(* CODESYS project mbc_Log4TC.library
   Title: Log4TC
   Version: 0.0.1
   Placeholder: Log4TC
   Company: mbc engineering GmbH

Project tree, tasks and I/O mapping:
  libraries: Base Interfaces, * (System); Tc2_Standard, * (Beckhoff Automation GmbH); Tc2_System, * (Beckhoff Automation GmbH); Tc2_Utilities, * (Beckhoff Automation GmbH)
  API/
    Full/
      function block FB_Logger [ST]: FB_init, LoggerContext
    Simple/
      function F_Log3 [ST]
      function F_Log3L [ST]
      function F_LogA3 [ST]
      function F_LogBuilder [ST]
      function F_LogLA3 [ST]
      interface I_LogBuilder: CreateLog, WithContextInt, WithIntArg, WithLogger, WithStringArg
    data type E_LogLevel
    function F_CallLogTask [ST]
    function F_LogContext [ST]
    interface I_ContextBuilder: Reset, WithInt
  GVLs/
    global variables Config
    global variables Const
    global variables GlobalVariables
  ITFs/
    interface I_LogEntryAdder: AddToLogEntry
  POUs/
    Utils/
      function F_DINT_TO_UINT_MAX [ST]
    function F_InternalLog [ST]
    function block FB_ContextBuilder [CFC]: _AddContext, _Copy, _RemoveContext, _Reset, _WriteByte, _WriteInt, AddToLogEntry, Reset, WithInt
    function block FB_Log4TcTask [CFC]: AddLog, Call, FB_init
    function block FB_LogEntry [CFC]: _BufferRemaining, _Copy, _Reset, _WriteArg, _WriteByte, _WriteDInt, _WriteInt, _WriteLInt, _WriteString, _WriteUDInt, _WriteUInt, AddAnyArg, AddBuffer, AddContext, AddTArg, End, GetBuffer, Start
  program Test [ST]
*)

// API/E_LogLevel
{attribute 'qualified_only'}
{attribute 'strict'}
TYPE E_LogLevel :
(
	eTrace 	:= 0,
	eDebug 	:= 1,
	eInfo	:= 2,
	eWarn	:= 3,
	eError	:= 4,
	eFatal	:= 5
) UINT;
END_TYPE

// GVLs/Config
{attribute 'qualified_only'}
VAR_GLOBAL CONSTANT
	eInternalLog		: E_LogLevel := E_LogLevel.eDebug;	(* min. log level for internal logging. *)
	nBufferLen 			: UINT := 8192;		(* Length of per task log buffer in bytes *)
END_VAR

// GVLs/Const
{attribute 'qualified_only'}
VAR_GLOBAL CONSTANT
	nAdsPort			: UINT := 16150; 
	nLogIndexGrp		: UINT := 1;
	nLogIndexOffs		: UINT := 1;
	
	sGlobalLogger		: STRING := '_GLOBAL_';		(* Global logger name for logger without logger input *)
END_VAR

// GVLs/GlobalVariables
{attribute 'qualified_only'}
VAR_GLOBAL
	aTaskLogger			: ARRAY[1..SIZEOF(TwinCAT_SystemInfoVarList._TaskInfo)/SIZEOF(PlcTaskSystemInfo)] OF FB_Log4TcTask;
END_VAR

// API/Full/FB_Logger
{attribute 'reflection'} 
FUNCTION_BLOCK FB_Logger
VAR_INPUT
	bExecute		: BOOL := TRUE;
	eLogLevel		: E_LogLevel;
	sMessage		: Tc2_System.T_MaxString;
	stArg1			: T_Arg := Tc2_Utilities.EMPTY_ARG_VALUE;
	stArg2			: T_Arg := Tc2_Utilities.EMPTY_ARG_VALUE;
	stArg3			: T_Arg := Tc2_Utilities.EMPTY_ARG_VALUE;
	stArg4			: T_Arg := Tc2_Utilities.EMPTY_ARG_VALUE;
	stArg5			: T_Arg := Tc2_Utilities.EMPTY_ARG_VALUE;	
	stArg6			: T_Arg := Tc2_Utilities.EMPTY_ARG_VALUE;	
	stArg7			: T_Arg := Tc2_Utilities.EMPTY_ARG_VALUE;	
	stArg8			: T_Arg := Tc2_Utilities.EMPTY_ARG_VALUE;	
	stArg9			: T_Arg := Tc2_Utilities.EMPTY_ARG_VALUE;	
	stArg10			: T_Arg := Tc2_Utilities.EMPTY_ARG_VALUE;	
	iContextBuilder	: I_ContextBuilder := 0;	
END_VAR
VAR
    {attribute 'instance-path'} 
    {attribute 'noinit'} // 'log4tc.log4Tc_Tester.MAIN.fbLog' bwz. 'log4tc.log4Tc_Tester.GVL.fbLog'
    sInstancePath	: T_MaxString; 	
	sLogger			: T_MaxString;
	fbLoggerContext	: FB_ContextBuilder;
END_VAR
VAR_TEMP
	fbLogEntry		: FB_LogEntry();
	fbSysTime		: Tc2_System.GETSYSTEMTIME;
	nTimestamp		: LINT;
	pBuffer			: PVOID;
	nBufferCount	: UINT;
	iLogEntryAdder	: I_LogEntryAdder;
END_VAR

IF bExecute THEN
	
	fbLogEntry.Start(
		pLogger		:= ADR(sLogger),
		pMessage 	:= ADR(sMessage),
		eLogLevel	:= eLogLevel,
		nTimeStampPlc := nTimestamp,
		nTimeStampClock := 0
	);
	
	fbLogEntry.AddTArg(1, stArg1);
	fbLogEntry.AddTArg(2, stArg2);
	fbLogEntry.AddTArg(3, stArg3);
	fbLogEntry.AddTArg(4, stArg4);
	fbLogEntry.AddTArg(5, stArg5);
	fbLogEntry.AddTArg(6, stArg6);
	fbLogEntry.AddTArg(7, stArg7);
	fbLogEntry.AddTArg(8, stArg8);
	fbLogEntry.AddTArg(9, stArg9);
	fbLogEntry.AddTArg(10, stArg10);
	
	//IF __QUERYINTERFACE(F_GetTaskContext(), iLogEntryAdder) THEN
		//iLogEntryAdder.AddToLogEntry(fbLogEntry);
	//END_IF
	
	fbLoggerContext.AddToLogEntry(fbLogEntry);
	
	IF iContextBuilder <> 0 AND __QUERYINTERFACE(iContextBuilder, iLogEntryAdder) THEN
		iLogEntryAdder.AddToLogEntry(fbLogEntry);
	END_IF
	
	// TODO instance path
	
	IF fbLogEntry.End() THEN
		// Add to buffer
		fbLogEntry.GetBuffer(
			pBuffer			=> pBuffer,
			nBufferCount	=> nBufferCount
		);
		GlobalVariables.aTaskLogger[GETCURTASKINDEXEX()].AddLog(pBuffer, nBufferCount);
	END_IF
END_IF

// reset arguments to default values
bExecute := TRUE;
stArg1 := Tc2_Utilities.EMPTY_ARG_VALUE;
stArg2 := Tc2_Utilities.EMPTY_ARG_VALUE;
stArg3 := Tc2_Utilities.EMPTY_ARG_VALUE;
stArg4 := Tc2_Utilities.EMPTY_ARG_VALUE;
stArg5 := Tc2_Utilities.EMPTY_ARG_VALUE;
stArg6 := Tc2_Utilities.EMPTY_ARG_VALUE;
stArg7 := Tc2_Utilities.EMPTY_ARG_VALUE;
stArg8 := Tc2_Utilities.EMPTY_ARG_VALUE;
stArg9 := Tc2_Utilities.EMPTY_ARG_VALUE;
stArg10 := Tc2_Utilities.EMPTY_ARG_VALUE;
iContextBuilder := 0;

METHOD FB_init : BOOL
VAR_INPUT
	bInitRetains : BOOL; // if TRUE, the retain variables are initialized (warm start / cold start)
	bInCopyCode : BOOL;  // if TRUE, the instance afterwards gets moved into the copy code (online change)
	sLogger		: T_MaxString;
END_VAR
THIS^.sLogger := sLogger;
END_METHOD

PROPERTY PUBLIC LoggerContext : I_ContextBuilder
GET
LoggerContext := fbLoggerContext;
END_GET
END_PROPERTY

END_FUNCTION_BLOCK

// API/I_ContextBuilder
INTERFACE I_ContextBuilder EXTENDS __System.IQueryInterface

METHOD Reset : I_ContextBuilder
VAR_INPUT
END_VAR
END_METHOD

METHOD WithInt : I_ContextBuilder
VAR_INPUT
	sName		: T_MaxString;
	nValue		: INT;
END_VAR
END_METHOD

END_INTERFACE

// POUs/FB_ContextBuilder
FUNCTION_BLOCK FB_ContextBuilder IMPLEMENTS I_ContextBuilder, I_LogEntryAdder
VAR CONSTANT
	nBufferSize			: UINT := 1024;
END_VAR
VAR
	aBuffer				: ARRAY[0..nBufferSize - 1] OF BYTE;	(* buffer for context variables *)
	nBufferCount		: UINT := 0;
	
	aContext			: ARRAY[0..19] OF UINT;
	nContextCount		: UINT(0..20) := 0;
END_VAR

METHOD PRIVATE _AddContext : BOOL
VAR_INPUT
END_VAR
IF nContextCount < 20 THEN
	aContext[nContextCount] := nBufferCount;
	nContextCount := nContextCount + 1;
	_AddContext := TRUE;
ELSE
	_AddContext := FALSE;
END_IF
END_METHOD

METHOD PRIVATE _Copy : BOOL
VAR_INPUT
	pSrc		: PVOID;
	nCount		: UINT;
END_VAR
IF (nBufferSize - nBufferCount) >= nCount THEN
	MEMCPY(ADR(aBuffer) + nBufferCount, pSrc, nCount);
	nBufferCount := nBufferCount + nCount;
	
	_Copy := TRUE;
ELSE
	_Copy := FALSE;
END_IF
END_METHOD

METHOD PRIVATE _RemoveContext : BOOL
VAR_INPUT
	refName		: REFERENCE TO Tc2_System.T_MaxString;
END_VAR
VAR
	nIdx		: UINT;
	nBufferOff	: UINT;
END_VAR
IF nContextCount > 0 THEN
	FOR nIdx := 0 TO nContextCount - 1 DO
		IF MEMCMP(ADR(refName), ADR(aBuffer) + aContext[nIdx], INT_TO_UDINT(LEN(refName) + 1)) = 0 THEN
			(* Found - remove entry and compact buffer *)
			IF (nIdx + 1) < nContextCount THEN
				// Move buffer data
				MEMMOVE(
					ADR(aBuffer) + aContext[nIdx], 
					ADR(aBuffer) + aContext[nIdx + 1], 
					nBufferCount - aContext[nIdx + 1]
				);
				
				nBufferOff := aContext[nIdx + 1] - aContext[nIdx];
				nBufferCount := nBufferCount - nBufferOff;
				
				// Move and change index
				WHILE (nIdx + 1) < nContextCount DO
					aContext[nIdx] := aContext[nIdx + 1] - nBufferOff;
					nIdx := nIdx + 1;
				END_WHILE
			END_IF

			nContextCount := nContextCount - 1;
			_RemoveContext := TRUE;
			RETURN;
		END_IF
	END_FOR
END_IF

_RemoveContext := FALSE;
END_METHOD

METHOD PRIVATE _Reset
VAR_INPUT
END_VAR
nBufferCount := 0;
nContextCount := 0;
END_METHOD

METHOD PRIVATE _WriteByte : BOOL
VAR_INPUT
	nValue		: BYTE;
END_VAR
_WriteByte := _Copy(ADR(nValue), SIZEOF(nValue));
END_METHOD

METHOD PRIVATE _WriteInt : BOOL
VAR_INPUT
	nValue		: INT;
END_VAR
_WriteInt := _Copy(ADR(nValue), SIZEOF(nValue));
END_METHOD

METHOD AddToLogEntry : BOOL
VAR_INPUT
	refLogEntry		: REFERENCE TO FB_LogEntry;
END_VAR
VAR
	nIdx			: UINT;
	bOk				: BOOL;
	nContextLen		: UINT;
END_VAR
nIdx := 0;
bOk := TRUE;
WHILE nIdx < nContextCount AND bOk DO
	IF (nIdx + 1) < nContextCount THEN
		nContextLen := aContext[nIdx + 1] - aContext[nIdx];
	ELSE
		nContextLen := nBufferCount - aContext[nIdx];
	END_IF
	
	refLogEntry.AddContext(ADR(aBuffer) + aContext[nIdx], nContextLen);
	
	nIdx := nIdx + 1;
END_WHILE 

AddToLogEntry := bOk;
END_METHOD

METHOD Reset : I_ContextBuilder
VAR_INPUT
END_VAR
_Reset();
Reset := THIS^;
END_METHOD

METHOD WithInt : I_ContextBuilder
VAR_INPUT
	sName	: Tc2_System.T_MaxString;
	nValue	: INT;
END_VAR
_RemoveContext(sName);

IF _AddContext() THEN
	_Copy(ADR(sName), INT_TO_UINT(LEN(sName) + 1));
	_WriteInt(E_ArgType.ARGTYPE_INT);
	_Copy(ADR(nValue), SIZEOF(nValue));
END_IF

WithInt := THIS^;
END_METHOD

END_FUNCTION_BLOCK

// ITFs/I_LogEntryAdder
INTERFACE I_LogEntryAdder EXTENDS __System.IQueryInterface

METHOD AddToLogEntry : BOOL
VAR_INPUT
	refLogEntry		: REFERENCE TO FB_LogEntry;
END_VAR
END_METHOD

END_INTERFACE

// POUs/FB_LogEntry
{attribute 'no_explicit_call' := 'no direct call necessary'} 
FUNCTION_BLOCK FB_LogEntry
VAR
	aBuffer				: ARRAY[1..Config.nBufferLen] OF BYTE;
	nBufferCount		: UINT;
	bError				: BOOL;
END_VAR

PROPERTY PRIVATE _BufferRemaining : UINT
GET
_BufferRemaining := SIZEOF(aBuffer) - nBufferCount;
END_GET
END_PROPERTY

METHOD PRIVATE _Copy
VAR_INPUT
	pSrc		: PVOID;
	nCount		: UINT;
END_VAR
IF NOT bError AND_THEN _BufferRemaining >= nCount THEN
	Tc2_System.MEMCPY(ADR(aBuffer) + nBufferCount, pSrc, nCount);
	nBufferCount := nBufferCount + nCount;
ELSE
	IF NOT bError THEN
		F_InternalLog(
			E_LogLevel.eWarn,
			'FB_LogEntry._Copy',
			'Error buffer overflow for log message (act=%d, new=%d)',
			Tc2_Utilities.F_UINT(nBufferCount),
			Tc2_Utilities.F_UINT(nCount),
			Tc2_Utilities.EMPTY_ARG_VALUE,
			Tc2_Utilities.EMPTY_ARG_VALUE
		);
	END_IF
	bError := TRUE;
END_IF
END_METHOD

METHOD PRIVATE _Reset
VAR_INPUT
END_VAR
nBufferCount := 0;
bError := FALSE;
END_METHOD

METHOD PRIVATE _WriteArg
VAR_INPUT
	stArg		: Tc2_Utilities.T_Arg;
END_VAR
VAR
	bOk			: BOOL;
END_VAR
_Copy(ADR(stArg.eType), SIZEOF(stArg.eType));

_Copy(stArg.pData, UDINT_TO_UINT(stArg.cbLen));
END_METHOD

METHOD PRIVATE _WriteByte 
VAR_INPUT
	nValue		: BYTE;
END_VAR
_Copy(ADR(nValue), SIZEOF(nValue));
END_METHOD

METHOD PRIVATE _WriteDInt
VAR_INPUT
	nValue		: DINT;
END_VAR
_Copy(ADR(nValue), SIZEOF(nValue));
END_METHOD

METHOD PRIVATE _WriteInt 
VAR_INPUT
	nValue		: INT;
END_VAR
_Copy(ADR(nValue), SIZEOF(nValue));
END_METHOD

METHOD PRIVATE _WriteLInt
VAR_INPUT
	nValue		: LINT;
END_VAR
_Copy(ADR(nValue), SIZEOF(nValue));
END_METHOD

METHOD PRIVATE _WriteString
VAR_INPUT
	pValue		: POINTER TO Tc2_Utilities.T_MaxString;
END_VAR
VAR
	nLen			: INT;
END_VAR
IF pValue <> 0 THEN
	nLen := Tc2_Standard.LEN(pValue^);
	IF nLen >= 0 AND nLen <= 255 THEN
		_WriteByte(INT_TO_BYTE(nLen)); 
		_Copy(ADR(pValue), INT_TO_UINT(nLen));
	ELSE
		// should not happen because T_MaxString is <= 255 bytes long
		bError := TRUE;
		F_InternalLog(
			E_LogLevel.eError,
			'FB_LogEntry._WriteString',
			'String longer than 255 bytes (actual=%d) - missin 0-byte?',
			Tc2_Utilities.F_INT(nLen),
			Tc2_Utilities.EMPTY_ARG_VALUE,
			Tc2_Utilities.EMPTY_ARG_VALUE,
			Tc2_Utilities.EMPTY_ARG_VALUE
		);
	END_IF
ELSE
		bError := TRUE;
		F_InternalLog(
			E_LogLevel.eError,
			'FB_LogEntry._WriteString',
			'String null pointer',
			Tc2_Utilities.EMPTY_ARG_VALUE,
			Tc2_Utilities.EMPTY_ARG_VALUE,
			Tc2_Utilities.EMPTY_ARG_VALUE,
			Tc2_Utilities.EMPTY_ARG_VALUE
		);
END_IF
END_METHOD

METHOD PRIVATE _WriteUDInt
VAR_INPUT
	nValue		: UDINT;
END_VAR
_Copy(ADR(nValue), SIZEOF(nValue));
END_METHOD

METHOD PRIVATE _WriteUInt 
VAR_INPUT
	nValue		: UINT;
END_VAR
_Copy(ADR(nValue), SIZEOF(nValue));
END_METHOD

METHOD INTERNAL AddAnyArg : BOOL
VAR_INPUT
	nArgNo		: BYTE;
	stArg		: ANY;
END_VAR
VAR
	bOk			: BOOL;
END_VAR
IF stArg.pValue = 0 THEN
	RETURN;
END_IF

_WriteByte(1); // Type 1: Argument follows
_WriteByte(nArgno);

CASE UDINT_TO_DINT(stArg.TypeClass) OF
	IBaseLibrary.TypeClass.TYPE_BOOL:
		_WriteInt(Tc2_Utilities.E_ArgType.ARGTYPE_BOOL);
		IF Tc2_Utilities.PBYTE_TO_BYTE(stArg.pValue) <> 0 THEN
			_WriteByte(1);
		ELSE
			_WriteByte(0);
		END_IF

	IBaseLibrary.TypeClass.TYPE_BYTE:
		_WriteInt(Tc2_Utilities.E_ArgType.ARGTYPE_BYTE);
		_Copy(stArg.pValue, SIZEOF(BYTE));
	
	IBaseLibrary.TypeClass.TYPE_WORD:
		_WriteInt(Tc2_Utilities.E_ArgType.ARGTYPE_WORD);
		_Copy(stArg.pValue, SIZEOF(WORD));		
	
	IBaseLibrary.TypeClass.TYPE_DWORD:
		_WriteInt(Tc2_Utilities.E_ArgType.ARGTYPE_DWORD);
		_Copy(stArg.pValue, SIZEOF(DWORD));		
	
	IBaseLibrary.TypeClass.TYPE_LWORD:
		_WriteInt(Tc2_Utilities.E_ArgType.ARGTYPE_LWORD);
		_Copy(stArg.pValue, SIZEOF(LWORD));
	
	IBaseLibrary.TypeClass.TYPE_SINT:
		_WriteInt(Tc2_Utilities.E_ArgType.ARGTYPE_SINT);
		_Copy(stArg.pValue, SIZEOF(SINT));
	
	IBaseLibrary.TypeClass.TYPE_INT:
		_WriteInt(Tc2_Utilities.E_ArgType.ARGTYPE_INT);
		_Copy(stArg.pValue, SIZEOF(INT));		
	
	IBaseLibrary.TypeClass.TYPE_DINT:
		_WriteInt(Tc2_Utilities.E_ArgType.ARGTYPE_DINT);
		_Copy(stArg.pValue, SIZEOF(DINT));		
	
	IBaseLibrary.TypeClass.TYPE_LINT:
		_WriteInt(Tc2_Utilities.E_ArgType.ARGTYPE_LARGE);
		_Copy(stArg.pValue, SIZEOF(LINT));		
	
	IBaseLibrary.TypeClass.TYPE_USINT:
		_WriteInt(Tc2_Utilities.E_ArgType.ARGTYPE_USINT);
		_Copy(stArg.pValue, SIZEOF(USINT));
	
	IBaseLibrary.TypeClass.TYPE_UINT:
		_WriteInt(Tc2_Utilities.E_ArgType.ARGTYPE_UINT);
		_Copy(stArg.pValue, SIZEOF(UINT));		
	
	IBaseLibrary.TypeClass.TYPE_UDINT:
		_WriteInt(Tc2_Utilities.E_ArgType.ARGTYPE_UDINT);
		_Copy(stArg.pValue, SIZEOF(UDINT));		
	
	IBaseLibrary.TypeClass.TYPE_ULINT:
		_WriteInt(Tc2_Utilities.E_ArgType.ARGTYPE_ULARGE);
		_Copy(stArg.pValue, SIZEOF(ULINT));		
	
	IBaseLibrary.TypeClass.TYPE_REAL:
		_WriteInt(Tc2_Utilities.E_ArgType.ARGTYPE_REAL);
		_Copy(stArg.pValue, SIZEOF(REAL));		
	
	IBaseLibrary.TypeClass.TYPE_LREAL:
		_WriteInt(Tc2_Utilities.E_ArgType.ARGTYPE_LREAL);
		_Copy(stArg.pValue, SIZEOF(LREAL));		
	
	IBaseLibrary.TypeClass.TYPE_STRING:
		_WriteInt(Tc2_Utilities.E_ArgType.ARGTYPE_STRING);
		_WriteString(stArg.pValue);

	//IBaseLibrary.TypeClass.TYPE_WSTRING:
		// TODO

	//IBaseLibrary.TypeClass.TYPE_TIME:
		//_WriteInt(Tc2_Utilities.E_ArgType.ARGTYPE_TIME);
		//_Copy(stArg.pValue, F_DINT_TO_UINT_MAX(stArg.diSize, SIZEOF(TIME)));

	//IBaseLibrary.TypeClass.TYPE_DATE:
		//_Copy(stArg.pValue, F_DINT_TO_UINT_MAX(stArg.diSize, SIZEOF(DATE)));

	//IBaseLibrary.TypeClass.TYPE_DATEANDTIME:
		//_Copy(stArg.pValue, F_DINT_TO_UINT_MAX(stArg.diSize, SIZEOF(Date_)));

	//IBaseLibrary.TypeClass.TYPE_TIMEOFDAY:
		//_Copy(stArg.pValue, F_DINT_TO_UINT_MAX(stArg.diSize, SIZEOF(TIMEOFDAY)));

	//IBaseLibrary.TypeClass.TYPE_ENUM:
		//_Copy(stArg.pValue, F_DINT_TO_UINT_MAX(stArg.diSize, 8));

	//IBaseLibrary.TypeClass.TYPE_LTIME:
		//_Copy(stArg.pValue, F_DINT_TO_UINT_MAX(stArg.diSize, SIZEOF(LTIME)));
		
	ELSE
		F_InternalLog(
			E_LogLevel.eWarn,
			'FB_LogEntry.AddAnyArg',
			'Unhandled ANY type=%d',
			Tc2_Utilities.F_UDINT(stArg.TypeClass),
			Tc2_Utilities.EMPTY_ARG_VALUE,
			Tc2_Utilities.EMPTY_ARG_VALUE,
			Tc2_Utilities.EMPTY_ARG_VALUE
		);
		// TODO maybe rollback and ignore argument or use replacement value (null)
		bError := TRUE;
END_CASE

AddAnyArg := NOT bError;
END_METHOD

METHOD INTERNAL AddBuffer
VAR_INPUT
	pBuffer			: PVOID;
	nBufferLen		: UINT;
END_VAR
_Copy(pBuffer, nBufferLen);
END_METHOD

METHOD PUBLIC AddContext
VAR_INPUT
	pBuffer			: PVOID;
	nBufferLen		: UINT;
END_VAR
_WriteByte(2); // Type 2: Context follows
_Copy(pBuffer, nBufferLen);
END_METHOD

METHOD INTERNAL AddTArg
VAR_INPUT
	nArgNo		: BYTE;
	stArg		: Tc2_Utilities.T_Arg;
END_VAR
VAR
	bOk			: BOOL;
END_VAR
IF stArg.eType = E_ArgType.ARGTYPE_UNKNOWN THEN
	RETURN;
END_IF

_WriteByte(1); // Type 1: Argument follows
_WriteByte(nArgNo);
_WriteArg(stArg);
END_METHOD

METHOD PUBLIC End : BOOL
_WriteByte(255);

End := NOT bError;
END_METHOD

METHOD PUBLIC GetBuffer : BOOL
VAR_OUTPUT
	pBuffer			: PVOID;
	nBufferCount	: UINT;
END_VAR
pBuffer := ADR(aBuffer);
nBufferCount := THIS^.nBufferCount;
END_METHOD

METHOD INTERNAL Start : BOOL
VAR_INPUT
	pLogger		: POINTER TO T_MaxString;
	pMessage		: POINTER TO T_MaxString;
	eLogLevel		: E_LogLevel;
	nTimeStampPlc	: LINT;
	nTimeStampClock	: LINT;
END_VAR
VAR
	fbSysTime		: Tc2_System.GETSYSTEMTIME;
	nTaskIndex		: DINT;
END_VAR
// Timestamp PLC
IF nTimestampPlc = 0 THEN
	fbSysTime();
	nTimeStampPlc := ULINT_TO_LINT(SHL(UDINT_TO_ULINT(fbSysTime.timeHiDW), 32) OR fbSysTime.timeLoDW);
END_IF

_Reset();

// Log-Entry Version
_WriteByte(1);

// Message
_WriteString(pMessage);

// Logger
_WriteString(pLogger);

// Level
_WriteUInt(eLogLevel);

// Timestamp PLC
_WriteLInt(nTimeStampPlc);

// Timestamp Clock
_WriteLInt(nTimeStampClock);

// Task Infos 
nTaskIndex := Tc2_System.GETCURTASKINDEXEX();
_WriteDInt(nTaskIndex);
_WriteString(ADR(TwinCAT_SystemInfoVarList._TaskInfo[nTaskIndex].TaskName));
_WriteUDInt(TwinCAT_SystemInfoVarList._TaskInfo[nTaskIndex].CycleCount);

// App Infos
_WriteString(ADR(TwinCAT_SystemInfoVarList._AppInfo.AppName));
_WriteString(ADR(TwinCAT_SystemInfoVarList._AppInfo.ProjectName));
_WriteUDInt(TwinCAT_SystemInfoVarList._AppInfo.OnlineChangeCnt);

Start := NOT bError;
END_METHOD

END_FUNCTION_BLOCK

// POUs/F_InternalLog
FUNCTION F_InternalLog : BOOL
VAR_INPUT
	eLogLevel 			: E_LogLevel;
	sContext			: Tc2_System.T_MaxString;
	sMessageFmt			: Tc2_System.T_MaxString;
	stArg1				: Tc2_Utilities.T_Arg;
	stArg2				: Tc2_Utilities.T_Arg;
	stArg3				: Tc2_Utilities.T_Arg;
	stArg4				: Tc2_Utilities.T_Arg;
END_VAR
VAR
	sOutputStr			: T_MaxString;
	fbFormatStr			: FB_FormatString;
	aBoolToByte			: ARRAY[1..4] OF BYTE;
	pBool				: POINTER TO BOOL;
END_VAR

IF eLogLevel < Config.eInternalLog THEN
	RETURN;
END_IF

CASE eLogLevel OF
	E_LogLevel.eTrace:
		sOutputStr := '[TRACE] ';
	E_LogLevel.eDebug:
		sOutputStr := '[DEBUG] ';
	E_LogLevel.eInfo:
		sOutputStr := '[INFO] ';
	E_LogLevel.eWarn:
		sOutputStr := '[WARN] ';
	E_LogLevel.eError:
		sOutputStr := '[ERROR] ';
	ELSE
		sOutputStr := '[FATAL] ';
END_CASE

IF LEN(sContext) > 0 THEN
	sOutputStr := CONCAT(sOutputStr, CONCAT(sContext, ' - '));
END_IF

IF stArg1.eType = E_ArgType.ARGTYPE_BOOL THEN
	pBool := stArg1.pData;
	aBoolToByte[1] := SEL(pBool^, 0, 1);
	stArg1 := F_BYTE(aBoolToByte[1]);
END_IF

IF stArg2.eType = E_ArgType.ARGTYPE_BOOL THEN
	pBool := stArg2.pData;
	aBoolToByte[2] := SEL(pBool^, 0, 1);
	stArg2 := F_BYTE(aBoolToByte[2]);
END_IF

IF stArg3.eType = E_ArgType.ARGTYPE_BOOL THEN
	pBool := stArg3.pData;
	aBoolToByte[3] := SEL(pBool^, 0, 1);
	stArg3 := F_BYTE(aBoolToByte[3]);
END_IF

IF stArg4.eType = E_ArgType.ARGTYPE_BOOL THEN
	pBool := stArg4.pData;
	aBoolToByte[4] := SEL(pBool^, 0, 1);
	stArg4 := F_BYTE(aBoolToByte[4]);
END_IF


fbFormatStr(
	sFormat := sMessageFmt,
	arg1 	:= stArg1,
	arg2	:= stArg2,
	arg3	:= stArg3,
	arg4	:= stArg4,
);

sOutputStr := CONCAT(sOutputStr, fbFormatStr.sOut);

ADSLOGSTR(ADSLOG_MSGTYPE_LOG, sOutputStr, '');

END_FUNCTION

// POUs/Utils/F_DINT_TO_UINT_MAX
FUNCTION F_DINT_TO_UINT_MAX : UINT
VAR_INPUT
	nValue			: DINT;
	nMaxValue		: UINT;
END_VAR

IF nValue < 0 THEN
	F_DINT_TO_UINT_MAX := 0;
ELSIF nValue > nMaxValue THEN
	F_DINT_TO_UINT_MAX := nMaxValue;
ELSE
	F_DINT_TO_UINT_MAX := DINT_TO_UINT(nValue);
END_IF

END_FUNCTION

// API/Simple/F_Log3
FUNCTION F_Log3 
VAR_INPUT
	eLogLevel		: E_LogLevel;
	sMessage		: T_MaxString;
	stArg1			: T_Arg;
	stArg2			: T_Arg;
	stArg3			: T_Arg;
END_VAR

END_FUNCTION

// API/Simple/F_Log3L
FUNCTION F_Log3L 
VAR_INPUT
	eLogLevel		: E_LogLevel;
	sLogger			: T_MaxString;
	sMessage		: T_MaxString;
	stArg1			: T_Arg;
	stArg2			: T_Arg;
	stArg3			: T_Arg;
END_VAR

END_FUNCTION

// API/Simple/F_LogA3
FUNCTION F_LogA3 
VAR_INPUT
	eLogLevel		: E_LogLevel;
	sMessage		: T_MaxString;
	aArg1			: ANY;
	aArg2			: ANY;
	aArg3			: ANY;
END_VAR
VAR
	fbLogEntry		: FB_LogEntry();
	pBuffer			: PVOID;
	nBufferCount	: UINT;	
END_VAR

F_LogLA3(eLogLevel, Const.sGlobalLogger, sMessage, aArg1, aArg2, aArg3);

END_FUNCTION

// API/Simple/F_LogLA3
FUNCTION F_LogLA3 
VAR_INPUT
	eLogLevel		: E_LogLevel;
	sLogger			: T_MaxString;
	sMessage		: T_MaxString;
	aArg1			: ANY;
	aArg2			: ANY;
	aArg3			: ANY;
END_VAR
VAR CONSTANT
	sGlobalLogger	: STRING := '_GLOBAL_';
END_VAR
VAR
	fbLogEntry		: FB_LogEntry();
	pBuffer			: PVOID;
	nBufferCount	: UINT;	
END_VAR

fbLogEntry.Start(
	pLogger			:= ADR(sGlobalLogger),
	pMessage		:= ADR(sMessage),
	eLogLevel		:= eLogLevel,
	nTimeStampPlc	:= 0,
	nTimeStampClock	:= 0
);

fbLogEntry.AddAnyArg(1, aArg1);
fbLogEntry.AddAnyArg(2, aArg2);
fbLogEntry.AddAnyArg(3, aArg3);

IF fbLogEntry.End() THEN
	// Add to task ring buffer
	fbLogEntry.GetBuffer(
		pBuffer			=> pBuffer,
		nBufferCount	=> nBufferCount
	);
	GlobalVariables.aTaskLogger[GETCURTASKINDEXEX()].AddLog(pBuffer, nBufferCount);
END_IF

END_FUNCTION

// API/Simple/F_LogBuilder
FUNCTION F_LogBuilder : I_LogBuilder
VAR_INPUT
	eLogLevel		: E_LogLevel;
	sMessages		: T_MaxString;
END_VAR

END_FUNCTION

// API/Simple/I_LogBuilder
INTERFACE I_LogBuilder

METHOD CreateLog
END_METHOD

METHOD WithContextInt : I_LogBuilder
VAR_INPUT
	sName		: T_MaxString;
	nValue		: INT;
END_VAR
END_METHOD

METHOD WithIntArg : I_LogBuilder
VAR_INPUT
	nValue		: INT;
END_VAR
END_METHOD

METHOD WithLogger : I_LogBuilder
VAR_INPUT
	sLogger		: T_MaxString;
END_VAR
END_METHOD

METHOD WithStringArg : I_LogBuilder
VAR_INPUT
	sValue		: T_MaxString;
END_VAR
END_METHOD

END_INTERFACE

// API/F_CallLogTask
FUNCTION F_CallLogTask

GlobalVariables.aTaskLogger[GETCURTASKINDEXEX()].Call();

END_FUNCTION

// API/F_LogContext
FUNCTION F_LogContext : I_ContextBuilder
VAR_STAT
	aTaskContext		: ARRAY[1..SIZEOF(TwinCAT_SystemInfoVarList._TaskInfo)/SIZEOF(PlcTaskSystemInfo)] OF FB_ContextBuilder;
END_VAR

F_LogContext := aTaskContext[Tc2_System.GETCURTASKINDEXEX()].Reset();

END_FUNCTION

// POUs/FB_Log4TcTask
(*
Main code of Log4TC which manages log messages of a single task.
*)
FUNCTION_BLOCK INTERNAL FB_Log4TcTask
VAR
	nTaskIndex			: DINT;
	fbRingBuffer		: Tc2_Utilities.FB_MemRingBufferEx;
	aBuffer				: ARRAY[1..Config.nBufferLen] OF BYTE;
	fbTaskContext		: FB_ContextBuilder;
END_VAR

METHOD INTERNAL AddLog : BOOL
VAR_INPUT
	pLogBuffer		: PVOID;
	nLogBufferLen	: UINT;
END_VAR
VAR
	nActTaskIndex		: DINT;
	bAddOk			: BOOL;
END_VAR
nActTaskIndex := Tc2_System.GETCURTASKINDEXEX();
IF nActTaskIndex = 0 OR nActTaskIndex <> nTaskIndex THEN
	F_InternalLog(
		E_LogLevel.eFatal,
		'Log4TcTask.AddLog',
		'Logger called in wrong task. Expected=%d Actual=%d',
		Tc2_Utilities.F_DINT(nTaskIndex),
		Tc2_Utilities.F_DINT(nActTaskIndex),
		Tc2_Utilities.EMPTY_ARG_VALUE,
		Tc2_Utilities.EMPTY_ARG_VALUE
	);
	AddLog := FALSE;
	RETURN;
END_IF

fbRingBuffer.A_AddTail(
	pBuffer 	:= ADR(aBuffer),
	cbBuffer 	:= SIZEOF(aBuffer),
	pWrite		:= pLogBuffer,
	cbWrite		:= nLogBufferLen,	
	bOk			=> bAddOk,
);

IF NOT bAddOk THEN
	F_InternalLog(
		E_LogLevel.eFatal,
		'Log4TcTask.AddLog',
		'Error adding log message to buffer. TaskIdx=%d MessageSize=%d BufferFree=%',
		Tc2_Utilities.F_DINT(nTaskIndex),
		Tc2_Utilities.F_UINT(nLogBufferLen),
		Tc2_Utilities.F_UDINT(fbRingBuffer.cbFree),
		Tc2_Utilities.EMPTY_ARG_VALUE
	);
ELSE
	F_InternalLog(
		E_LogLevel.eTrace,
		'Log4TcTask.AddLog',
		'Adding log message to buffer. TaskIdx=%d MessageSize=%d BufferFree=%',
		Tc2_Utilities.F_DINT(nTaskIndex),
		Tc2_Utilities.F_UINT(nLogBufferLen),
		Tc2_Utilities.F_UDINT(fbRingBuffer.cbFree),
		Tc2_Utilities.EMPTY_ARG_VALUE
	);	
END_IF 

AddLog := bAddOk;
END_METHOD

(*
Should be called regularly in the same task as its instance was
declared.
*)
METHOD INTERNAL Call
VAR
	nMessageCount		: UINT;
END_VAR
VAR_INST
	nState				: UINT;
	nActTaskIndex		: DINT;
	aSendBuffer			: ARRAY[1..Config.nBufferLen] OF BYTE;		(* Buffer for send data *)
	nSendBufferLen		: UDINT;
	bContinue			: BOOL;
	fbAdsWriteMsg		: Tc2_System.ADSWRITE:=(PORT:=Const.nAdsPort);
END_VAR
nActTaskIndex := Tc2_System.GETCURTASKINDEXEX();
IF nTaskIndex = 0 AND nActTaskIndex > 0 THEN
	nTaskIndex := nActTaskIndex;
ELSIF nTaskIndex <> nActTaskIndex OR nActTaskIndex = 0 THEN
	F_InternalLog(
		E_LogLevel.eFatal,
		'Log4TcTask.Call',
		'Log4Tc Task called in wrong task (expected=%d actual=%d)',
		F_DINT(nTaskIndex),
		F_DINT(nActTaskIndex),
		Tc2_Utilities.EMPTY_ARG_VALUE,
		Tc2_Utilities.EMPTY_ARG_VALUE
	);
	RETURN;
END_IF

CASE nState OF
	0: // Init
		nSendBufferLen := 0;
		nState := 10;
		
	10: // Wait for log entry; add them to the send buffer
		nMessageCount := 0;
		REPEAT
			fbRingBuffer.A_GetHead(
				pBuffer 	:= ADR(aBuffer),
				cbBuffer 	:= SIZEOF(aBuffer),
			);
			
			IF fbRingBuffer.bOk AND (SIZEOF(aSendBuffer) - nSendBufferLen) >= fbRingBuffer.cbRead THEN
				MEMCPY(ADR(aSendBuffer) + nSendBufferLen, fbRingBuffer.pRead, fbRingBuffer.cbRead);
				nSendBufferLen := nSendBufferLen + fbRingBuffer.cbRead;
				
				fbRingBuffer.A_FreeHead(
					pBuffer 	:= ADR(aBuffer),
					cbBuffer 	:= SIZEOF(aBuffer),
				);
				
				nMessageCount := nMessageCount + 1;
				bContinue := TRUE;
			ELSE
				bContinue := FALSE;
			END_IF
		UNTIL
			NOT bContinue
		END_REPEAT;

		IF nSendBufferLen > 0 THEN
			F_InternalLog(
				E_LogLevel.eDebug,
				'FB_Log4TcTask.Call',
				'Sending %d message with size %d.',
				Tc2_Utilities.F_UINT(nMessageCount),
				Tc2_Utilities.F_UDINT(nSendBufferLen),
				Tc2_Utilities.EMPTY_ARG_VALUE,
				Tc2_Utilities.EMPTY_ARG_VALUE
			);	
		
			fbAdsWriteMsg(WRITE:=FALSE);
			fbAdsWriteMsg(
				WRITE	:= TRUE,
				IDXGRP 	:= Const.nLogIndexGrp,
				IDXOFFS := Const.nLogIndexOffs,
				LEN		:= nSendBufferLen,
				SRCADDR	:= ADR(aSendBuffer),
			);
		
			nState := 20;
		END_IF
		
	20: // Wait for sent data
		fbAdsWriteMsg();
		IF NOT fbAdsWriteMsg.BUSY THEN
			IF fbAdsWriteMsg.ERR THEN
				F_InternalLog(
					E_LogLevel.eFatal,
					'Log4TcTask.Call',
					'Error sending log message to handler. task=%d adsErrId=%d',
					F_DINT(nTaskIndex),
					F_UDINT(fbAdsWriteMsg.ERRID),
					Tc2_Utilities.EMPTY_ARG_VALUE,
					Tc2_Utilities.EMPTY_ARG_VALUE
				);
			ELSE
				F_InternalLog(
					E_LogLevel.eDebug,
					'FB_Log4TcTask.Call',
					'Message successfully sent.',
					Tc2_Utilities.EMPTY_ARG_VALUE,
					Tc2_Utilities.EMPTY_ARG_VALUE,
					Tc2_Utilities.EMPTY_ARG_VALUE,
					Tc2_Utilities.EMPTY_ARG_VALUE
				);	
			END_IF
			
			nSendBufferLen := 0;
			nState := 10;
		END_IF
	
END_CASE
END_METHOD

METHOD FB_init : BOOL
VAR_INPUT
	bInitRetains : BOOL; // if TRUE, the retain variables are initialized (warm start / cold start)
	bInCopyCode : BOOL;  // if TRUE, the instance afterwards gets moved into the copy code (online change)
END_VAR
fbRingBuffer.A_Reset
(
	pBuffer 	:= ADR(aBuffer),
	cbBuffer 	:= SIZEOF(aBuffer),
);
END_METHOD

END_FUNCTION_BLOCK

// Test
PROGRAM Test
VAR
	fbLogger		: FB_Logger('mbc4Log.Test');
	nInt			: INT;
	sStr			: STRING;
	fFloat			: REAL;
END_VAR

// Einfaches Logging
F_Log3(
	E_LogLevel.eInfo, 
	'Log Message Arg={structuredArg} Arg={1} Arg=%s', 
	F_StringEx('Arg 1'),
	F_StringEx('Arg 2'),
	F_StringEx('Arg 3')
);

F_LogA3(
	E_LogLevel.eError,
	'Log Message Arg={structuredArg} Arg={1} Arg=%s',
	nInt,
	sStr,
	fFloat
);

// Einfaches Logging mit expliziten Logger
F_Log3L(
	E_LogLevel.eInfo, 
	'mbc4Log.Test',
	'Log Message Arg={structuredArg} Arg={1} Arg=%s', 
	F_StringEx('Arg 1'),
	F_StringEx('Arg 2'),
	F_StringEx('Arg 3')
);

// Einfaches Logging mit Builder
F_LogBuilder(E_LogLevel.eError, 'Log Message Arg={structuredArg} Arg={1} Arg=%s')
	.WithIntArg(42).WithStringArg('Arg 2').WithStringArg('Arg 3')
	.WithLogger('mbc4Log.Test')
	.WithContextInt('id', 42)
	.CreateLog();

fbLogger(
	eLogLevel 		:= E_LogLevel.eInfo, 
	sMessage 		:='Log Message Arg={structuredArg} Arg={1} Arg=%s', 
	stArg1 			:= F_StringEx('Arg 1'),
	stArg2 			:= F_StringEx('Arg 2'),
	stArg3 			:= F_StringEx('Arg 3'),
	iContextBuilder	:= F_LogContext().WithInt('id', 42)
);

END_PROGRAM
